{attribute 'qualified_only'}
{attribute 'strict'}
{attribute 'to_string'}
TYPE ETransport :
(
	Off:=0,
	Init := 1,
	Ready := 2,
	Production := 3,
	Producing := 4,
	Done := 5
);
END_TYPE

(* stored: Version 1.1.0.1
   DUT ETransport: Id {250f902b-59c7-4f97-a9b8-082e176b5988} *)
